// TIA Portal V18 export
FUNCTION "ST10_Input" : Void   // FC1001, LAD
{ S7_Optimized_Access := 'FALSE' }
VERSION : 0.1
// 注：本程序用来处理需要滤波，延时、计算的输入信号
// stored: AutoNumber false, IsIECCheckEnabled false, SetENOAutomatically false, UDAEnableTagReadback false
BEGIN

REGION Network 1 (SCL): HMI信号映射 / HMI signal mapping
   "ST10_SysInput".HMI_Button.ControlOn := "iHMI Control On";
   //"ST350_SysInput".HMI_Button.ControlOff:=
   "ST10_SysInput".HMI_Button.MachineStart := "iHMI Machine Start";
   "ST10_SysInput".HMI_Button.MachineStop := "iHMI Machine Stop";
   "ST10_SysInput".HMI_Button.ResetButton := "iHMI ResetButton";
   "ST10_SysInput".HMI_Button."Manual/Auto" := "iHMI Manual/Auto";
   "ST10_SysInput".HMI_Button.SafetyGateUnlock := "iHMI Safety Gate Unlock";
   "ST10_SysInput".HMI_Button."E-Stop" :=  "iHMI E-Stop";
END_REGION

REGION Network 2 (SCL): Sys IO Image
   "ST10_SysInput".Sys.iCircuitBreakerOK1 := "iCircuit Breaker OK_1";
   "ST10_SysInput".Sys.iCircuitBreakerOK2 := "iCircuit Breaker OK_2";
   "ST10_SysInput".Sys.iPressure:= "iPressure";
END_REGION

REGION Network 3 (SCL): iE-StopPB
   "ST10_SysInput"."iE-StopPB"[1] := "iE_StopButton2_A01";
   "ST10_SysInput"."iE-StopPB"[2] := "iE_StopButton3_A02";
   "ST10_SysInput"."iE-StopPB"[3] := "iE_StopButton4_H";
   "ST10_SysInput"."iE-StopPB"[4] := "iE_StopButton5_J";
   "ST10_SysInput"."iE-StopPB"[5] := "iE_StopButton6_K";
   "ST10_SysInput"."iE-StopPB"[6] := "iE_StopButton7_L";
   "ST10_SysInput"."iE-StopPB"[7] := "iH_StopButton";
   "ST10_SysInput"."iE-StopPB"[8] := "iJ_StopButton";
   "ST10_SysInput"."iE-StopPB"[9] := "iK_StopButton";
END_REGION

REGION Network 4 (SCL): iSafetyGatFeedBack
   (*
   "ST350_SysInput".iSafetyGatFeedBack[1] := "iSafety door Locking FeedBack_1";
   "ST350_SysInput".iSafetyGatFeedBack[2] := "iSafety door Locking FeedBack_2";
   "ST350_SysInput".iSafetyGatFeedBack[3] := "iSafety door Locking FeedBack_3";
   "ST350_SysInput".iSafetyGatFeedBack[4] := "iSafety door Locking FeedBack_4";
   "ST350_SysInput".iSafetyGatFeedBack[5] := "iSafety door Locking FeedBack_5";
   "ST350_SysInput".iSafetyGatFeedBack[6] := "iSafety door Locking FeedBack_6";
   "ST350_SysInput".iSafetyGatFeedBack[7] := "iSafety door Locking FeedBack_7";
   "ST350_SysInput".iSafetyGatFeedBack[8] := "iSafety door Locking FeedBack_8";
   *)
END_REGION

REGION Network 5 (SCL): iSafetydoorLockingFeedBack
   "ST10_SysInput".iSafetydoorLockingFeedBack[1] := "iSafety door Locking FeedBack_1";
   "ST10_SysInput".iSafetydoorLockingFeedBack[2] := "iSafety door Locking FeedBack_2";
   "ST10_SysInput".iSafetydoorLockingFeedBack[3] := "iSafety door Locking FeedBack_3";
   "ST10_SysInput".iSafetydoorLockingFeedBack[4] := "iSafety door Locking FeedBack_4";
   "ST10_SysInput".iSafetydoorLockingFeedBack[5] := "iSafety door Locking FeedBack_5";
   "ST10_SysInput".iSafetydoorLockingFeedBack[6] := "iSafety door Locking FeedBack_6";
   "ST10_SysInput".iSafetydoorLockingFeedBack[7] := "iSafety door Locking FeedBack_7";
   "ST10_SysInput".iSafetydoorLockingFeedBack[8] := "iSafety door Locking FeedBack_8";
END_REGION

REGION Network 6 (SCL): iSafetydoorLockingFeedBack
   "ST10_SysInput".iMaterieldoorLockingFeedBack[1] := "iMateriel Door Locking FeedBack_H1";
   "ST10_SysInput".iMaterieldoorLockingFeedBack[2] := "iMateriel Door Locking FeedBack_H2";
   "ST10_SysInput".iMaterieldoorLockingFeedBack[3] := "iMateriel Door Locking FeedBack_J1";
   "ST10_SysInput".iMaterieldoorLockingFeedBack[4] := "iMateriel Door Locking FeedBack_J2";
   "ST10_SysInput".iMaterieldoorLockingFeedBack[5] := "iMateriel Door Locking FeedBack_K1";
   "ST10_SysInput".iMaterieldoorLockingFeedBack[6] := "iMateriel Door Locking FeedBack_K2";
   "ST10_SysInput".iMaterieldoorLockingFeedBack[7] := "iMateriel Door Locking FeedBack_L1";
END_REGION
END_FUNCTION
